Fanuc KAREL source: kd_tree.klc

PROGRAM class_name
%NOBUSYLAMP
%COMMENT = 'kd tree'
%NOLOCKGROUP
%NOPAUSE = COMMAND + TPENABLE + ERROR

%define EPSILON 0.001

-- declare type
%include define_type.m

%defeval BASE_CLASSNAME class_name

%include errors.klt
%include systemlib.types.klt
%include binary_tree.c.klt
%include binary_tree.klt

%include kd_tree.klt
define_kd_types(KDTREE_QUERY_TYPE,class_name,KDTREE_COMPARE_TYPE)

%define BASE_CLASSNAME class_name

%ifdef USER_DEFINED_TYPES
%mode push
%mode quote "$"
%eval $%include USER_DEFINED_TYPES$
%mode pop
%endif

--hash to keep track of sorted and filtered data
%include hashpath.klt
hash_header_define(HASH_CLASS_NAME)
t_hash(hashname,hval_def,HASH_CLASS_NAME)

VAR
  this : PATH pathheader = HDR_BST, nodedata = T_BST
  data : PATH nodedata = KDTREE_DATA_TYPE
  hmap : PATH pathheader = t_linear_hsh, nodedata = hashname
  traverse : PATH nodedata = t_INTEGER
  current : INTEGER
  query : PATH nodedata = KDTREE_QUERY_TYPE
  frm : XYZWPR
  query_flag : BOOLEAN

%include errors.klh
%from strings.klh %import i_to_s, r_to_s, rarr_to_s, iarr_to_s, pose_to_s, vec_to_s, joint_to_s
%from math.klh %import ceil, manhattan_dist, norm, norm2

--hash table object
define_hash(HASH_CLASS_NAME,KD_CONFIG_FILE)

%defeval class_name BASE_CLASSNAME

%include kd_tree.klh
%include kd_tree.private.klh
--include user defined members
define_kd_members(class_name)

--private

ROUTINE clear_
  VAR
    i : INTEGER
    status : INTEGER
  BEGIN
    i = PATH_LEN(this)
    WHILE PATH_LEN(this) > 0 DO
		  DELETE_NODE(this,i,status)
      CHK_STAT(status)
      i = i - 1
	  ENDWHILE

    this.root = 0
  END clear_

ROUTINE clear_data
  VAR
    i : INTEGER
    status : INTEGER
  BEGIN
    i = PATH_LEN(d)
    WHILE PATH_LEN(d) > 0 DO
		  DELETE_NODE(d,i,status)
      CHK_STAT(status)
      i = i - 1
	  ENDWHILE
  END clear_data

ROUTINE reset_generator
  VAR
    i : INTEGER
    status : INTEGER
  BEGIN
    current = 0

    i = PATH_LEN(traverse)
    WHILE PATH_LEN(traverse) > 0 DO
		  DELETE_NODE(traverse,i,status)
      CHK_STAT(status)
      i = i - 1
	  ENDWHILE
  END reset_generator

ROUTINE clear_query
  VAR
    i : INTEGER
    status : INTEGER
  BEGIN
    i = PATH_LEN(query)
    WHILE PATH_LEN(query) > 0 DO
		  DELETE_NODE(query,i,status)
      i = i - 1
	  ENDWHILE
  END clear_query

ROUTINE new_node
  VAR
    i, status : INTEGER
  BEGIN
    IF idx > PATH_LEN(this) THEN
      FOR i = PATH_LEN(this)+1 TO idx DO
        APPEND_NODE(this, status)
        this[i].left = 0
        this[i].right = 0
      ENDFOR
    ENDIF
  END new_node

ROUTINE tree_comparator
  VAR
    r1, r2 : KDTREE_COMPARE_TYPE
    lconv, rconv : KDTREE_VALUE_TYPE
  BEGIN
    lconv = INV((frm)):l_val.KDTREE_NODE_NAME
    rconv = INV((frm)):r_val.KDTREE_NODE_NAME
    SELECT axs OF
      CASE(1):
        r1 = lconv.x ; r2 = rconv.x ;
      CASE(2):
        r1 = lconv.y ; r2 = rconv.y ;
      CASE(3):
        r1 = lconv.z ; r2 = rconv.z ;
      ELSE:
    ENDSELECT

    IF r1 > r2 THEN
      RETURN(GREATER_THAN)
    ENDIF
    IF r1 < r2 THEN
      RETURN(LESS_THAN)
    ENDIF
    IF r1 = r2 THEN
      RETURN(EQUAL_TO)
    ENDIF

    RETURN(0)
  END tree_comparator

ROUTINE inhypersphere
  VAR
    lconv, rconv : KDTREE_VALUE_TYPE
  BEGIN
    lconv = INV((frm)):point.KDTREE_NODE_NAME
    rconv = INV((frm)):plane.KDTREE_NODE_NAME
    SELECT axs OF
      CASE(1):
        -- check overlap on left subtree
        IF (lconv.x - dist) <= rconv.x THEN
          RETURN(TRUE)
        -- check overlap on right subtree
        ELSE IF (lconv.x + dist) > rconv.x THEN
          RETURN(TRUE)
        ENDIF
        ENDIF
      CASE(2):
        -- check overlap on left subtree
        IF (lconv.y - dist) <= rconv.y THEN
          RETURN(TRUE)
        -- check overlap on right subtree
        ELSE IF (lconv.y + dist) > rconv.y THEN
          RETURN(TRUE)
        ENDIF
        ENDIF
      CASE(3):
        -- check overlap on left subtree
        IF (lconv.z - dist) <= rconv.z THEN
          RETURN(TRUE)
        -- check overlap on right subtree
        ELSE IF (lconv.z + dist) > rconv.z THEN
          RETURN(TRUE)
        ENDIF
        ENDIF
      ELSE:
    ENDSELECT

    RETURN(FALSE)

  END inhypersphere

ROUTINE bubblesort
  VAR
    i,j : INTEGER
    n : INTEGER
    swap : KDTREE_DATA_TYPE
  BEGIN
    n = high
    FOR i=low TO high DO
      FOR j=low TO n-1 DO
        IF tree_comparator(list[j], list[j+1], axs) = LESS_THAN THEN
          swap = (list[j+1])
          list[j+1] = (list[j])
          list[j] = swap
        ENDIF
      ENDFOR
      n = n - 1
    ENDFOR
  END bubblesort

ROUTINE build_tree
  VAR
    idx : INTEGER
    mid : INTEGER
    b : BOOLEAN
  BEGIN
    IF data_start > data_end THEN
      new_node(data_end)
      RETURN(0)
    ENDIF

    bubblesort(data, data_start, data_end, (depth MOD DIMENSIONS) + 1)
    mid = TRUNC((data_start + data_end)/2)

    --find mid in hash table
    b = `HASH_CLASS_NAME`__get(user_string(data[mid]), idx, hmap)

    IF NOT b THEN
      karelError(INVALID_INDEX,'Could not find hash '+ vec_to_s(data[mid].v,',') +' while building kd tree', ER_ABORT)
    ENDIF

    IF this.root = 0 THEN
      this.root = idx
    ENDIF

    new_node(idx)
    this[idx].right = build_tree(data_start, mid-1, depth+1)
    this[idx].left = build_tree(mid+1, data_end, depth+1)

    IF (this[idx].right = idx) THEN this[idx].right = 0 ; ENDIF
    IF (this[idx].left = idx) THEN this[idx].left = 0 ; ENDIF

    RETURN(idx)

  END build_tree

ROUTINE inorder
  VAR
    status : INTEGER
  BEGIN
    IF idx > 0 THEN
      inorder((this[idx].left))
      APPEND_NODE(traverse, status)
      traverse[PATH_LEN(traverse)].v = idx
      inorder((this[idx].right))
    ENDIF
  END inorder

ROUTINE preorder
  VAR
    status : INTEGER
  BEGIN
    IF idx > 0 THEN
      APPEND_NODE(traverse, status)
      traverse[PATH_LEN(traverse)].v = idx
      preorder((this[idx].left))
      preorder((this[idx].right))
    ENDIF
  END preorder

ROUTINE postorder
  VAR
    status : INTEGER
  BEGIN
    IF idx > 0 THEN
      preorder((this[idx].left))
      preorder((this[idx].right))
      APPEND_NODE(traverse, status)
      traverse[PATH_LEN(traverse)].v = idx
    ENDIF
  END postorder

ROUTINE minmaxUtil
  VAR
    n1, n2 : INTEGER
  BEGIN
    -- evaluate down the left hand side of the tree if current depth
    -- is the evaluation axis
    IF (dim = (depth MOD DIMENSIONS) + 1) THEN
      SELECT mn_mx OF
        CASE(LESS_THAN):
          IF this[root].left = 0 THEN RETURN(root) ; ENDIF
          n1 = minmaxUtil((this[root].left), depth+1, dim, mn_mx)
        ELSE:
          IF this[root].right = 0 THEN RETURN(root) ; ENDIF
          n1 = minmaxUtil((this[root].right), depth+1, dim, mn_mx)
      ENDSELECT

      IF tree_comparator(data[n1], data[root], dim) = mn_mx THEN
        RETURN(n1)
      ENDIF
    ENDIF

    -- If current dimension is different than evaluation axis
    -- minimum can be anywhere in this subtree
    IF this[root].left = 0 THEN
      n1 = root
    ELSE
      n1 = minmaxUtil((this[root].left), depth+1, dim, mn_mx)
    ENDIF
    IF this[root].right = 0 THEN
      n2 = root
    ELSE
      n2 = minmaxUtil((this[root].right), depth+1, dim, mn_mx)
    ENDIF

    IF tree_comparator(data[n1], data[n2], dim) = mn_mx THEN
      IF tree_comparator(data[n1], data[root], dim) = mn_mx THEN
        RETURN(n1)
      ELSE
        RETURN(root)
      ENDIF
    ELSE
      IF tree_comparator(data[n2], data[root], dim) = mn_mx THEN
        RETURN(n2)
      ELSE
        RETURN(root)
      ENDIF
    ENDIF
  END minmaxUtil

ROUTINE kNNUtil
  VAR
    dist : KDTREE_COMPARE_TYPE
    i, status : INTEGER
    inserted : BOOLEAN
  BEGIN
    IF (root = 0) THEN
      RETURN
    ENDIF
    IF (NOT inhypersphere(query[1].value, point, data[root], (depth MOD DIMENSIONS)+1)) THEN
      RETURN
    ENDIF

    -- append node to query list
    IF query_flag OR query_filter(point, data[root]) THEN
      i = 1
      inserted = FALSE
      dist = distance(point, data[root])
      WHILE((i<=PATH_LEN(query)) AND (NOT inserted)) DO
        IF dist < query[i].value THEN
          INSERT_NODE(query, i, status)
          query[i].idx = root
          query[i].value = dist
          DELETE_NODE(query, PATH_LEN(query), status)
          inserted = TRUE
        ENDIF
        i = i + 1
      ENDWHILE
    ENDIF

    -- visit subtrees is most promising order:
    IF tree_comparator(point, data[root], (depth MOD DIMENSIONS)+1) = LESS_THAN THEN
      kNNUtil((this[root].left), depth+1, point)
      kNNUtil((this[root].right), depth+1, point)
    ELSE
      kNNUtil((this[root].right), depth+1, point)
      kNNUtil((this[root].left), depth+1, point)
    ENDIF

    RETURN

  END kNNUtil

ROUTINE rNNUtil
  VAR
    dist : KDTREE_COMPARE_TYPE
    i, status : INTEGER
    inserted : BOOLEAN
  BEGIN
    IF (root = 0) THEN
      RETURN
    ENDIF
    IF (NOT inhypersphere(query[1].value, point, data[root], (depth MOD DIMENSIONS)+1)) THEN
      RETURN
    ENDIF

    dist = distance(point, data[root])
    -- append node to query list
    IF (dist < radius) AND (query_flag OR query_filter(point, data[root])) THEN
      i = 1
      inserted = FALSE
      WHILE((i<=PATH_LEN(query)) AND (NOT inserted)) DO
        IF dist < query[i].value THEN
          INSERT_NODE(query, i, status)
          query[i].idx = root
          query[i].value = dist
          inserted = TRUE
        ENDIF
        i = i + 1
      ENDWHILE
    ENDIF

    -- visit subtrees is most promising order:
    IF tree_comparator(point, data[root], (depth MOD DIMENSIONS)+1) = LESS_THAN THEN
      rNNUtil((this[root].left), depth+1, (radius), point)
      rNNUtil((this[root].right), depth+1, (radius), point)
    ELSE
      rNNUtil((this[root].right), depth+1, (radius), point)
      rNNUtil((this[root].left), depth+1, (radius), point)
    ENDIF

    RETURN

  END rNNUtil

--public

ROUTINE clear
  VAR
    i : INTEGER
    status : INTEGER
  BEGIN
    clear_
    clear_data(data)
    reset_generator
    clear_query

    current = 0
    query_flag = FALSE
  END clear

ROUTINE create
  VAR
    i : INTEGER
    ret : INTEGER
    status : INTEGER
    b : BOOLEAN
  BEGIN
    clear
    frm = coord_frame
    query_flag = FALSE

    --copy data
    COPY_PATH(kd_data, 0, 0, data, status)

    --index original data in hash table
    `HASH_CLASS_NAME`__init(hmap)
    FOR i=1 TO PATH_LEN(data) DO
      b = `HASH_CLASS_NAME`__put(user_string(data[i]), i, hmap)
      IF NOT b THEN
        karelError(INVALID_INDEX,'Could not hash index:' + i_to_s(i) + ' in kd tree', ER_ABORT)
      ENDIF
    ENDFOR

    --build kd tree. data will be sorted.
    ret = build_tree(1, PATH_LEN(data), 0)

    --copy original unsorted data
    COPY_PATH(kd_data, 0, 0, data, status)

    --deallocate hash
    `HASH_CLASS_NAME`__destructor(hmap)

  END create

%ifdef INCLUDE_FILTER
ROUTINE create_filtered
  VAR
    i : INTEGER
    ret : INTEGER
    status : INTEGER
    b : BOOLEAN
  BEGIN
    clear
    frm = coord_frame
    query_flag = FALSE

    --index original data in hash table
    `HASH_CLASS_NAME`__init(hmap)
    FOR i=1 TO PATH_LEN(kd_data) DO
      b = `HASH_CLASS_NAME`__put(user_string(kd_data[i]), i, hmap)
      IF NOT b THEN
        karelError(INVALID_INDEX,'Could not hash index:' + i_to_s(i) + ' in kd tree', ER_ABORT)
      ENDIF
    ENDFOR

    --filter data
    filter(kd_data, data)

    --build kd tree. data will be sorted.
    ret = build_tree(1, PATH_LEN(data), 0)

    --copy original unsorted data
    COPY_PATH(kd_data, 0, 0, data, status)

    --deallocate hash
    `HASH_CLASS_NAME`__destructor(hmap)

  END create_filtered
%endif

ROUTINE new_generator
  BEGIN
    reset_generator

    SELECT typ OF
      CASE(IN_ORDER):
        inorder(this.root)
      CASE(PRE_ORDER):
        preorder(this.root)
      CASE(POST_ORDER):
        postorder(this.root)
      ELSE:
    ENDSELECT

  END new_generator

ROUTINE next
  BEGIN
    current = current + 1
    RETURN(data[traverse[current].v])
  END next

ROUTINE print
  VAR
    i : INTEGER
    nde : KDTREE_DATA_TYPE
  BEGIN
    new_generator(typ)

    WRITE TPDISPLAY(CR)
    FOR i=1 TO PATH_LEN(traverse) DO
      nde = next
      user_print(nde)
      WRITE TPDISPLAY(CR)
    ENDFOR
  END print

ROUTINE print_query
  VAR
    i : INTEGER
    nde : KDTREE_DATA_TYPE
  BEGIN
    WRITE TPDISPLAY(CR)
    FOR i=1 TO PATH_LEN(query) DO
      WRITE('p[', query[i].idx, ']: ')
      user_print(data[query[i].idx])
      WRITE(' d: ', query[i].value::5::2)
      WRITE TPDISPLAY(CR)
    ENDFOR
  END print_query

ROUTINE copy_data
  VAR
    status : INTEGER
  BEGIN
    COPY_PATH(data, 0, 0, out_list, status)
  END copy_data

ROUTINE get_query
  VAR
    i, status : INTEGER
  BEGIN
    FOR i=1 TO PATH_LEN(query) DO
      APPEND_NODE(out_list, status)
      out_list[PATH_LEN(out_list)].KDTREE_NODE_NAME = data[query[i].idx].KDTREE_NODE_NAME
    ENDFOR
  END get_query

ROUTINE get_query_arr
  VAR
    i, status : INTEGER
  BEGIN
    IF ARRAY_LEN(out_arr) < PATH_LEN(query) THEN
      karelError(ARR_LEN_MISMATCH,'output array is not large enough to contain query', ER_ABORT)
    ENDIF

    FOR i=1 TO PATH_LEN(query) DO
      out_arr[i] = data[query[i].idx].KDTREE_NODE_NAME
    ENDFOR
  END get_query_arr

ROUTINE get_query_idx
  VAR
    i, j, status : INTEGER
%ifndef MAX_NEIGHBORS
%define MAX_NEIGHBORS 5
%endif
    neigh : ARRAY[MAX_NEIGHBORS] OF KDTREE_QUERY_TYPE
  BEGIN
    IF ARRAY_LEN(neigh) < PATH_LEN(query) THEN
      karelError(ARR_LEN_MISMATCH,'Cant export query. Increase MAX_NEIGHBORS for get_query_idx.', ER_ABORT)
    ENDIF

    FOR i=1 TO PATH_LEN(query) DO
      neigh[i] = query[i]
    ENDFOR

    RETURN(neigh)
  END get_query_idx

ROUTINE enable_search_filter
  BEGIN
    query_flag = FALSE
  END enable_search_filter

ROUTINE disable_search_filter
  BEGIN
    query_flag = TRUE
  END disable_search_filter

ROUTINE findmin
  BEGIN
    RETURN(data[minmaxUtil(this.root, 0, dimension, LESS_THAN)])
  END findmin

ROUTINE findmax
  BEGIN
    RETURN(data[minmaxUtil(this.root, 0, dimension, GREATER_THAN)])
  END findmax

ROUTINE kth_nearest_neighbors
  VAR
    i, status : INTEGER
  BEGIN
    clear_query
    --fill query with kth nodes. Set 1st index for insert
    FOR i=1 TO k DO
      APPEND_NODE(query, status)
      query[i].idx = 0
      query[i].value = 0
    ENDFOR
    query[1].value = KDTREE_MAX_DIST

    kNNUtil(this.root, 0, point)

  END kth_nearest_neighbors

ROUTINE kNN_brute_force
  VAR
    i,j : INTEGER
    status : INTEGER
    dist : KDTREE_COMPARE_TYPE
    inserted : BOOLEAN
%ifdef INCLUDE_FILTER
    b : BOOLEAN
%endif
  BEGIN
%ifdef INCLUDE_FILTER
  --index original data in hash table
  `HASH_CLASS_NAME`__init(hmap)
  FOR i=1 TO PATH_LEN(list) DO
    b = `HASH_CLASS_NAME`__put(user_string(list[i]), i, hmap)
    IF NOT b THEN
      karelError(INVALID_INDEX,'Could not hash index:' + i_to_s(i) + ' in kd tree', ER_ABORT)
    ENDIF
  ENDFOR

  --filter data
  clear_data(data)
  filter(list, data)
%else
    --copy data into object
    COPY_PATH(list, 0, 0, data, status)
%endif

    clear_query
    --fill query with kth nodes. Set 1st index for insert
    FOR i=1 TO k DO
      APPEND_NODE(query, status)
      query[i].idx = 0
      query[i].value = 0
    ENDFOR
    query[1].value = KDTREE_MAX_DIST

    FOR i=1 TO PATH_LEN(data) DO
      -- append node to query list
      IF query_flag OR query_filter(point, data[i]) THEN
        j = 1
        inserted = FALSE
        dist = distance(point, data[i])
        WHILE((j<=PATH_LEN(query)) AND (NOT inserted)) DO
          IF dist < query[j].value THEN
            INSERT_NODE(query, j, status)
%ifdef INCLUDE_FILTER
            b = `HASH_CLASS_NAME`__get(user_string(data[i]), query[j].idx, hmap)
%else
            query[j].idx = i
%endif
            query[j].value = dist
            DELETE_NODE(query, PATH_LEN(query), status)
            inserted = TRUE
          ENDIF
          j = j + 1
        ENDWHILE
      ENDIF
    ENDFOR

%ifdef INCLUDE_FILTER
    --deallocate hash
    `HASH_CLASS_NAME`__destructor(hmap)
%endif

    -- return query
  END kNN_brute_force

ROUTINE radius_nearest_neighbors
  VAR
    i, status : INTEGER
  BEGIN
    clear_query

    APPEND_NODE(query, status)
    query[1].idx = 0
    query[1].value = KDTREE_MAX_DIST

    rNNUtil(this.root, 0, (radius), point)

    DELETE_NODE(query, PATH_LEN(query), status)

  END radius_nearest_neighbors

ROUTINE rNN_brute_force
  VAR
    i,j : INTEGER
    status : INTEGER
    dist : KDTREE_COMPARE_TYPE
    inserted : BOOLEAN
%ifdef INCLUDE_FILTER
    b : BOOLEAN
%endif
  BEGIN

%ifdef INCLUDE_FILTER
  --index original data in hash table
  `HASH_CLASS_NAME`__init(hmap)
  FOR i=1 TO PATH_LEN(list) DO
    b = `HASH_CLASS_NAME`__put(user_string(list[i]), i, hmap)
    IF NOT b THEN
      karelError(INVALID_INDEX,'Could not hash index:' + i_to_s(i) + ' in kd tree', ER_ABORT)
    ENDIF
  ENDFOR

  --filter data
  clear_data(data)
  filter(list, data)
%else
    --copy data into object
    COPY_PATH(list, 0, 0, data, status)
%endif

    clear_query

    --dummy placement node
    APPEND_NODE(query, status)
    query[1].idx = 0
    query[1].value = KDTREE_MAX_DIST

    FOR i=1 TO PATH_LEN(data) DO
      dist = distance(point, data[i])
      -- append node to query list
      IF (dist < radius) AND (query_flag OR query_filter(point, data[i])) THEN
        j = 1
        inserted = FALSE
        WHILE((j<=PATH_LEN(query)) AND (NOT inserted)) DO
          IF dist < query[j].value THEN
            INSERT_NODE(query, j, status)
%ifdef INCLUDE_FILTER
            b = `HASH_CLASS_NAME`__get(user_string(data[i]), query[j].idx, hmap)
%else
            query[j].idx = i
%endif
            query[j].value = dist
            inserted = TRUE
          ENDIF
          j = j + 1
        ENDWHILE
      ENDIF
    ENDFOR

    --remove last node, as it is only a dummy placement
    DELETE_NODE(query, PATH_LEN(query), status)

%ifdef INCLUDE_FILTER
    --deallocate hash
    `HASH_CLASS_NAME`__destructor(hmap)
%endif

    -- return query

  END rNN_brute_force

BEGIN
END class_name
